Staubli VAL3: chkDrivesFault.pgx

program chkDrivesFault()
  local num l_i
begin
  //检查电机是否有错误
  //以下情况表明电机出现错误:
  //错误标志位；
  bNoDrivesFault=true
  for l_i=0 to nAxesSum-1
    if bDrvFault[l_i]!=(diFault[l_i]==true) and (!bDrvFault[l_i])
      sMsg="第"+toString("",l_i+1)+"轴控制器报错"
      popUpMsg(sMsg)
      logMsg(sMsg)
    endIf
    bDrvFault[l_i]=(diFault[l_i]==true)
    bNoDrivesFault=bNoDrivesFault and !bDrvFault[l_i]
  endFor
end
